# EPICS autosave request: iocBoot/sioc-bc1b-bl01/blen_manual.req
file "common.req" AREA=BC1B,POS=850,INST=0
file "common.req" AREA=BC1B,POS=850,INST=1
file "pyro.req" AREA=BC1B,POS=850,INST=0
file "pyro.req" AREA=BC1B,POS=850,INST=1
